// TIA Portal V17 export
// export: Created 2024-06-19T09:47:14.7155746Z, ExportSetting WithDefaults, DisplayName Totally Integrated Automation Portal, DisplayVersion V17, DisplayName TIA Portal Openness, DisplayVersion V17, DisplayName TIA Portal Version Control Interface, DisplayVersion V17, DisplayName STEP 7 Professional, DisplayVersion V17, DisplayName STEP 7 Safety, DisplayVersion V17, DisplayName WinCC Professional, DisplayVersion V17
VAR_GLOBAL   // PLC tag table "St0_Out"
   IO_Verrou_PorteEntree AT %Q0.0 : Bool;   // Verrouillage : Porte d'entrée
   IO_Verrou_PorteSortie AT %Q0.1 : Bool;   // Verrouillage : Porte de sortie
   IO_Verrou_PorteVision AT %Q0.2 : Bool;   // Verrouillage : Porte maintenance vision façade
   IO_Verrou_PorteArriere AT %Q0.3 : Bool;   // Verrouillage : Porte maintenance arrière machine
   IO_Ouverture_PorteEntree AT %Q0.4 : Bool;   // Ouverture : Porte d'entrée
   IO_Ouverture_PorteSortie AT %Q0.5 : Bool;   // Ouverture : Porte de sortie
   IO_LED_Rouge AT %Q0.6 : Bool;   // Colonne lumineuse : Rouge
   IO_LED_Orange AT %Q0.7 : Bool;   // Colonne lumineuse : Orange
   IO_LED_Vert AT %Q1.0 : Bool;   // Colonne lumineuse : Vert
   IO_LED_Bleu AT %Q1.1 : Bool;   // Colonne lumineuse : Bleu
END_VAR
